FUNCTION_BLOCK DS_TrajectoryController IMPLEMENTS ITcIoUdpProtocolRecv
//aus Sicht GW3, Input: von GW2 zu Gw3, output: von GW3 zu GW2
VAR_INPUT
	wpListeRec: ARRAY[0...100] OF RobotPoseSimple;
	wpListeCirc: ARRAY[0...100] OF RobotPoseSimple;
END_VAR
VAR_OUTPUT
	fahren: BOOL := 0;		//1 = fahren
	amZiel: BOOL := 0;		//1 = am Ziel
END_VAR
VAR
	RechteckX: ARRAY[0...10] OF LREAL := [1000,3000,5000,5000,5000,3000,1000,1000,1000,-1];
	RechteckY: ARRAY[0...10] OF LREAL := [1000,1000,1000,1500,2000,2000,2000,1500,1000,-1];
	RechteckTheta: LREAL := pi/2;
	KreisX: ARRAY[0...10] OF LREAL := [4000,4200,4500,4700,5000,4700,4500,4200,4000,-1];
	KreisY: ARRAY[0...10] OF LREAL := [1500,1200,1000,1200,1500,1700,2000,1700,1500,-1];
	KreisTheta: LREAL := pi;
	randomParameter: INT := 0;
END_VAR

//fahren ohne Kollision
wpListeRec := ArrayToStruct(RechteckX,RechteckY, RechteckTheta);

WHILE fahren <> 1 DO
	randomParameter := 1;
END_WHILE;

WHILE amZiel <> 1 DO
	randomParameter := 2;
END_WHILE;

wpListeCirc := ArrayToStruct(RechteckX,RechteckY, RechteckTheta);

WHILE fahren <> 1 DO
	randomParameter := 3;
END_WHILE;

WHILE amZiel <> 1 DO
	randomParameter := 4;
END_WHILE;


//Rechteck
	//1000,1000,0
	//3000,1000,0
	//5000,1000,90
	//5000,1500,90
	//5000,2000,180
	//3000,2000,180
	//1000,2000,-90
	//1000,1500,-90
	//1000,1000,0 
	
//Kreis
	//4000, 1500, -45
	//4500, 1000, 45
	//5000, 1500, 135
	//4500, 2000, -135

{attribute 'TcTypeSystem'}
{attribute 'no-analysis'}
{attribute 'c++_compatible'}
{attribute 'minimal_input_size' := '4'}
{attribute 'pack_mode' := '4'}
{warning 'Methodenimplementierung hinzufügen'}
METHOD ReceiveData : HRESULT
VAR_INPUT
	ipAddr	: UDINT;
	udpDestPort	: UINT;
	udpSrcPort	: UINT;
	nData	: UDINT;
	pData	: PVOID;
	pVlan	: POINTER TO ETYPE_VLAN_HEADER := 0;
END_VAR
END_METHOD

{attribute 'TcTypeSystem'}
{attribute 'no-analysis'}
{attribute 'c++_compatible'}
{attribute 'minimal_input_size' := '4'}
{attribute 'pack_mode' := '4'}
{warning 'Methodenimplementierung hinzufügen'}
METHOD TcAddRef : UDINT
END_METHOD

{attribute 'TcTypeSystem'}
{attribute 'no-analysis'}
{attribute 'c++_compatible'}
{attribute 'minimal_input_size' := '4'}
{attribute 'pack_mode' := '4'}
{warning 'Methodenimplementierung hinzufügen'}
METHOD TcQueryInterface : HRESULT
VAR_INPUT
	iid	: REFERENCE TO IID;
	pipItf	: POINTER TO PVOID;
END_VAR
END_METHOD

{attribute 'TcTypeSystem'}
{attribute 'no-analysis'}
{attribute 'c++_compatible'}
{attribute 'minimal_input_size' := '4'}
{attribute 'pack_mode' := '4'}
{warning 'Methodenimplementierung hinzufügen'}
METHOD TcRelease : UDINT
END_METHOD

END_FUNCTION_BLOCK

(* stored: Version 1.1.0.1, ProductVersion 3.1.4024.11
   POU DS_TrajectoryController: Id {088ef7f9-632e-414f-83fe-772780584ea7}, SpecialFunc None
   Method ReceiveData: Id {876ceff4-21e0-48e4-b506-a672d857e671}
   Method TcAddRef: Id {a724e14b-b97a-4d35-99c5-b7db2456f759}
   Method TcQueryInterface: Id {4a0ce0e0-df2b-49ce-8b7a-3628d707309a}
   Method TcRelease: Id {2252b447-c0dc-4c4b-90fa-58df4d2c4c07} *)
